FUNCTION TryConvert_WORD_TO_DATE : BOOL
VAR_INPUT
	in : WORD;
	out : REFERENCE TO DATE;
END_VAR

out := WORD_TO_DATE(in);
TryConvert_WORD_TO_DATE := TRUE;

END_FUNCTION

(* stored: Version 1.1.0.1, ProductVersion 3.1.4024.12
   POU TryConvert_WORD_TO_DATE: Id {d487abd7-9bb0-4aa3-b77a-998c5a78797e}, SpecialFunc None *)
